// TwinCAT 3 PLC project TcIotOcppChargingStationPlc
// Title: TwinCAT IoT OCPP Charging Station Sample
// Company: Beckhoff Automation GmbH & Co. KG
// ProjectVersion: 1.0.0.0
// ProgramVersion: 3.1.4026.10
// libraries:
//   Tc2_Standard, * (Beckhoff Automation GmbH)
//   Tc2_System, * (Beckhoff Automation GmbH)
//   Tc2_Utilities, * (Beckhoff Automation GmbH)
//   Tc3_Module, * (Beckhoff Automation GmbH)
//   Tc3_OCPP, * (Beckhoff Automation GmbH)
// project tree:
//   GVLs/ VAR_OCPP.TcGVL, VAR_Param.TcGVL
//   / PlcTask.TcTTO
//   POUs/ FB_ConnectorSim.TcPOU, MAIN.TcPOU
//   POUs/OCPP/ FB_Connector.TcPOU, FB_ConnectorMeter.TcPOU, FB_MeterValue.TcPOU, FB_SampleValue.TcPOU, FB_Station.TcPOU, FB_StationMeter.TcPOU
// real-time tasks:
//   TASK PlcTask: cycle T#10ms, priority 20, ADS port 350

CONFIGURATION TcIotOcppChargingStationPlc
    RESOURCE PLC ON TwinCAT3
        TASK PlcTask(INTERVAL := T#10ms, PRIORITY := 20);
        PROGRAM MAIN WITH PlcTask : MAIN;
    END_RESOURCE
END_CONFIGURATION

// ---- GVLs/VAR_OCPP.TcGVL
{attribute 'qualified_only'}
VAR_GLOBAL
	stClientParam : ST_OCPP1_ClientParam := (
		//nOID : OTCID := 0; // ObjectID of the TcIotOcpp Client Object (0 to create a new instance).
		nTaskOID := 0, // ObjectId of the Task whose shall execute the client (0 to use I/O Idle Task)
		sHost := 'localhost', // Defines the server-address by host-name, domain-name or IP-address.
		nPort := 8080, // Defines the server-port.
		sPath := 'ocpp', // Defines the server-path.
		sIdentity := 'Test01', // Defines the client-identity (and user-id).
		eAuthMode := E_OCPP1_AuthenticationMode.Basic, // Defines an optional authentication-mode.
		sAuthKey := 'abcdef', // Defines an optional authentication key.
		eEncryptionMode := E_OCPP_EncryptionMode.None, // Defines an optional encryption mode.
		eTraceLevel := TcTraceLevel.tlVerbose); // Defines the maximum trace level of ADS log messages.

	stOptions : ST_OCPP1_ClientOptions := (
		bAllowOfflineTxForUnknownId := FALSE, // Whether Unknown Offline Authorization is enabled.
		bAuthListEnabled := FALSE, // Whether the Local Authorization List is enabled.
		bAuthCacheEnabled := FALSE, // Whether the Authorization Cache is enabled.
		bLocalAuthOffline := FALSE, // Whether the Charge Point, when offline, will start a transaction for locally-authorized identifiers.
		bLocalPreAuth := FALSE); // Whether the Charge Point, when online, will start a transaction for locally-authorized identifiers without waiting for an response from the Central System.

	stSettings : ST_OCPP1_ClientSettings := (
		nTransactionMessageAttempts := 5, // How often the Charge Point should try to submit a transaction-related message when the Central System fails to process it.
		nTransactionMessageRetryInterval := 5); // [s] How long the Charge Point should wait before resubmitting a transaction-related message that the Central System failed to process.

	stBootInfo : ST_OCPP1_ClientBootInfo := (
		sChargePointModel := 'TcIotOcppStation', // Required. This contains a value that identifies the model of the ChargePoint.
		sChargePointVendor := 'Beckhoff Automation', // Required. This contains a value that identifies the vendor of the ChargePoint.
		sChargeBoxSerialNumber := '', // Optional. This contains a value that identifies the serial number of the Charge Box inside the Charge Point.
		sChargePointSerialNumber := '', // Optional. This contains a value that identifies the serial number of the Charge Point.
		sFirmwareVersion := '', // Optional. This contains the firmware version of the Charge Point.
		sMeterSerialNumber := '', // Optional. This contains the serial number of the main electrical meter of the Charge Point.
		sMeterType := ''); // Optional. This contains the type of the main electrical meter of the Charge Point.

	fCurrentOffered1 : REAL := 16.0; // [A] current offered on every phace of connector (11kW)
	fCurrentOffered2 : REAL := 12.0; // [A] current offered on every phace of connector (8kW)
END_VAR

// ---- GVLs/VAR_Param.TcGVL
{attribute 'qualified_only'}
VAR_GLOBAL CONSTANT
	tSamplePeriodic : TIME := T#30S; // Interval of sample periodic meter values in FB_ConnectorMeter
	tSampleClock : TIME := T#60S; // Interval of sample clock meter values in FB_StationMeter
END_VAR

// ---- POUs/MAIN.TcPOU
PROGRAM MAIN
VAR
	// Station/Connectors
	fbStation : FB_Station(stParam := VAR_OCPP.stClientParam);
	fbConnector1 : FB_Connector(nConnectorId := 1, fbStation := fbStation);
	fbConnector2 : FB_Connector(nConnectorId := 2, fbStation := fbStation);
	// MeterValues/SampledValues
	fbStationMeter : FB_StationMeter(fbStation := fbStation);
	fbConnector1Meter : FB_ConnectorMeter(nConnectorId := 1, fbStation := fbStation);
	fbConnector2Meter : FB_ConnectorMeter(nConnectorId := 2, fbStation := fbStation);
	// Simulation
	fbConnector1Sim : FB_ConnectorSim;
	fbConnector2Sim : FB_ConnectorSim;
END_VAR

fbStation.Execute();

fbStationMeter.Execute(fbStation := fbStation);
fbConnector1Meter.Execute(fbConnector := fbConnector1, fCurrentOffered := VAR_OCPP.fCurrentOffered1);
fbConnector2Meter.Execute(fbConnector := fbConnector2, fCurrentOffered := VAR_OCPP.fCurrentOffered2);

fbConnector1Sim(fbConnector := fbConnector1, fCurrentOffered := VAR_OCPP.fCurrentOffered1);
fbConnector2Sim(fbConnector := fbConnector2, fCurrentOffered := VAR_OCPP.fCurrentOffered2);

END_PROGRAM

// ---- POUs/OCPP/FB_Station.TcPOU
FUNCTION_BLOCK FB_Station
VAR_OUTPUT
	bBusy : BOOL;
	bError : BOOL;
	eState : E_OCPP1_ChargePointStatus := E_OCPP1_ChargePointStatus.Available;
	eErrorState : E_OCPP1_ChargePointStatus := E_OCPP1_ChargePointStatus.None;
END_VAR
VAR
	// client
	_oClient : FB_OCPP1_Client(0);
	// connectors
	_arrConnectors : ARRAY[1..Param_OCPP.nConnectorCount] OF POINTER TO FB_Connector;
	_nConnectorCnt : UDINT;
	_nConnectorMax : UDINT;
	// configuration
	_fbConfiguration : FB_OCPP1_Configuration;
	// charging profile
	_fbChargingProfile : FB_OCPP1_ChargingProfile;
	_arrCharging : ARRAY[1..Param_OCPP.nConnectorCount] OF BOOL;
	// reset
	_fbTcRestart : TC_Restart;
	_fbOsRestart : NT_Reboot;
	
	bTest: BOOL;
END_VAR
VAR PERSISTENT
	_bAvailable : BOOL := TRUE;
END_VAR

METHOD INTERNAL AddConnector : BOOL
VAR_INPUT
	nConnectorId : UDINT;
	pConnector : POINTER TO FB_Connector;
END_VAR
IF nConnectorId < 1 OR nConnectorId > Param_OCPP.nConnectorCount THEN
	RETURN; // invalid connector id!
END_IF

IF pConnector = 0 THEN
	RETURN; // invalid pointer to connector!
END_IF

IF _arrConnectors[nConnectorId] <> 0 THEN
	RETURN; // connector id already used!
END_IF

_arrConnectors[nConnectorId] := pConnector;

_nConnectorCnt := _nConnectorCnt + 1;
IF nConnectorId > _nConnectorMax THEN _nConnectorMax := nConnectorId; END_IF

AddConnector := TRUE;
END_METHOD

PROPERTY Available : BOOL
GET
Available := _oClient.IsConnected
	AND eState <> E_OCPP1_ChargePointStatus.Unavailable
	AND eState <> E_OCPP1_ChargePointStatus.Faulted;
END_GET
END_PROPERTY

PROPERTY INTERNAL Client : POINTER TO FB_OCPP1_Client
GET
Client := ADR(_oClient);
END_GET
END_PROPERTY

METHOD PRIVATE Configuration : BOOL
VAR_STAT
	sValue : T_OCPP1_ConfigValue;
	nValue : UDINT;
END_VAR
IF _fbConfiguration.HasChanged(E_OCPP1_ConfigKey.HeartbeatInterval) THEN
	sValue := _fbConfiguration.GetValue(E_OCPP1_ConfigKey.HeartbeatInterval);
	_oClient.HeartbeatInterval := UDINT_TO_TIME(STRING_TO_UDINT(sValue)*1000);
END_IF
END_METHOD

METHOD Execute : BOOL
VAR
	nIdx : UDINT;
	eAction : E_OCPP1_Action;
	mPeriod : ST_OCPP1_ChargingSchedulePeriod;
END_VAR
_oClient.Execute(TRUE);
bBusy := _oClient.bBusy;

IF _oClient.bError THEN
	bError := TRUE;
	eErrorState := eState;
	eState := E_OCPP1_ChargePointStatus.Faulted;
END_IF

// ================================================================================
// Execute Connectors and apply Charging Profile

FOR nIdx := 1 TO Param_OCPP.nConnectorCount DO
	_arrConnectors[nIdx]^.Execute();
	_arrCharging[nIdx] := _arrConnectors[nIdx]^.bCharging;
END_FOR

_fbChargingProfile.Execute(_arrCharging, _oClient);

FOR nIdx := 1 TO Param_OCPP.nConnectorCount DO
	_fbChargingProfile.GetCurrentPeriod(nIdx, mPeriod);
	_arrConnectors[nIdx]^.SetChargingSchedulePeriod(mPeriod);
END_FOR

// ================================================================================
// State machine of Charging Station

CASE eState OF
	E_OCPP1_ChargePointStatus.Available: // Operative
		IF NOT _bAvailable THEN
			eState := E_OCPP1_ChargePointStatus.Unavailable;
		END_IF

	E_OCPP1_ChargePointStatus.Unavailable: // Inoperative, e.g. as result of a ChangeAvailability command.
		IF _bAvailable THEN
			eState := E_OCPP1_ChargePointStatus.Available;
		END_IF

	E_OCPP1_ChargePointStatus.Faulted: // Inoperative, when charger or connector has reported an error and is not available for energy delivery.

ELSE
	bError := TRUE;
	eErrorState := eState;
	eState := E_OCPP1_ChargePointStatus.Faulted;
END_CASE

// ================================================================================
// Send status of Charging Station

SendStatusNotification();

// ================================================================================
// Receive requests from Management System

IF _oClient.PollRequest(eAction => eAction) THEN
	CASE eAction OF
		// Core
		E_OCPP1_Action.RemoteStartTransaction:
			RecvRemoteStartTransaction();
		E_OCPP1_Action.RemoteStopTransaction:
			RecvRemoteStopTransaction();
		E_OCPP1_Action.ChangeAvailability:
			RecvChangeAvailability();
		E_OCPP1_Action.UnlockConnector:
			RecvUnlockConnector();
		E_OCPP1_Action.ChangeConfiguration:
			_fbConfiguration.Execute(_oClient);
		E_OCPP1_Action.GetConfiguration:
			_fbConfiguration.Execute(_oClient);
		//E_OCPP1_Action.ClearCache
		E_OCPP1_Action.Reset:
			RecvReset();
		// Remote Trigger
		E_OCPP1_Action.TriggerMessage:
			RecvTriggerMessage();
		// Reservation
		E_OCPP1_Action.ReserveNow:
			RecvReserveNow();
		E_OCPP1_Action.CancelReservation:
			RecvReserveCancel();
		// Smart Charging
		E_OCPP1_Action.SetChargingProfile:
			_fbChargingProfile.Execute(_arrCharging, _oClient);
		E_OCPP1_Action.GetCompositeSchedule:
			_fbChargingProfile.Execute(_arrCharging, _oClient);
		E_OCPP1_Action.ClearChargingProfile:
			_fbChargingProfile.Execute(_arrCharging, _oClient);
		// Authentication
		//E_OCPP1_Action.GetLocalListVersion
		//E_OCPP1_Action.SendLocalList
		// Firmware
		//E_OCPP1_Action.GetDiagnostics
		//E_OCPP1_Action.UpdateFirmware
		// Vendor
		E_OCPP1_Action.DataTransfer:
			RecvDataTransfer();
		// Security
		//E_OCPP1_Action.ExtendedTriggerMessage
		//E_OCPP1_Action.GetLog
		//E_OCPP1_Action.GetInstalledCertificateIds
		//E_OCPP1_Action.CertificateSigned
		//E_OCPP1_Action.SignCertificate
		//E_OCPP1_Action.InstallCertificate
		//E_OCPP1_Action.DeleteCertificate
		//E_OCPP1_Action.SignedUpdateFirmware
	ELSE
		// TODO response
	END_CASE
END_IF

// ================================================================================
// Additional functionalities

_fbTcRestart(RESTART := FALSE);
_fbOsRestart(START := FALSE);

Configuration();
SendDataTransfer();
END_METHOD

METHOD FB_Init : BOOL
VAR_INPUT
	bInitRetains : BOOL; // if TRUE, the retain variables are initialized (warm start / cold start)
	bInCopyCode : BOOL;  // if TRUE, the instance afterwards gets moved into the copy code (online change)

	stParam :  REFERENCE TO ST_OCPP1_ClientParam; // Parameter to define the OCPP WebSocket connection.
END_VAR
IF bInCopyCode THEN RETURN; END_IF

IF NOT __ISVALIDREF(stParam) THEN RETURN; END_IF

FB_Init := Init(stParam);
END_METHOD

METHOD Init : BOOL
VAR_INPUT
	stParam : REFERENCE TO ST_OCPP1_ClientParam; // Parameter to define the OCPP WebSocket connection.
END_VAR
Init := _oClient.Init(stParam);

_oClient.InitOptions(VAR_OCPP.stOptions);
_oClient.InitSettings(VAR_OCPP.stSettings);
_oClient.InitBootInfo(VAR_OCPP.stBootInfo);

_fbConfiguration.InitStandard();
_fbConfiguration.InitKeyValue(E_OCPP1_ConfigKey.HeartbeatInterval, UDINT_TO_STRING(TIME_TO_UDINT(_oClient.HeartbeatInterval)/1000), FALSE);
END_METHOD

PROPERTY IsConnected : BOOL
GET
IsConnected := _oClient.IsConnected;
END_GET
END_PROPERTY

METHOD PRIVATE RecvChangeAvailability : BOOL
VAR_STAT
	hRecvId : T_OCPP_MessageId;
	nConnectorId : UDINT; // The id of the connector for which availability needs to change.
	eType : E_OCPP1_AvailabilityType; // This contains the type of availability change that the Charge Point should perform.
	eStatus : E_OCPP1_AvailabilityStatus; // This indicates whether the Charge Point is able to perform the availability change.
END_VAR
// Central System can request a Charge Point to change its availability
// - A Charge Point is considered available ("operative") when it is charging or ready for charging
// - A Charge Point is considered unavailable when it does not allow any charging
IF _oClient.RecvChangeAvailability(hMessageId=> hRecvId, nConnectorId=> nConnectorId, eType=> eType) THEN
	eStatus := E_OCPP1_AvailabilityStatus.Rejected;
	IF nConnectorId = 0 THEN
		CASE eType OF
			E_OCPP1_AvailabilityType.Operative:
				_bAvailable := TRUE;
				eStatus := E_OCPP1_AvailabilityStatus.Accepted;
			E_OCPP1_AvailabilityType.Inoperative:
				_bAvailable := FALSE;
				eStatus := E_OCPP1_AvailabilityStatus.Accepted;
		END_CASE
		FOR nConnectorId := 1 TO _nConnectorMax DO
			IF _arrConnectors[nConnectorId] <> 0 THEN
				_arrConnectors[nConnectorId]^.ChangeAvailability(eType:= eType, eStatus=> eStatus);
			END_IF
		END_FOR
	ELSE
		IF _arrConnectors[nConnectorId] <> 0 THEN
			IF _arrConnectors[nConnectorId]^.ChangeAvailability(eType:= eType, eStatus=> eStatus) THEN
		 		eStatus := E_OCPP1_AvailabilityStatus.Accepted;
			END_IF
		END_IF
	END_IF
	_oClient.RespChangeAvailability(hMessageId:= hRecvId, eStatus:= eStatus);
END_IF
END_METHOD

METHOD RecvDataTransfer : BOOL
VAR_STAT
	hRecvId : T_OCPP_MessageId;
	sVendorId : STRING(255); 
	sMessageId : STRING(63); 
	sData : T_OCPP1_DataTransferData; 
END_VAR
IF _oClient.RecvDataTransfer(hMessageId => hRecvId, sVendorId=> sVendorId, sMessageId=> sMessageId, sData := sData) THEN
	IF sVendorId <> 'Beckhoff Automation' THEN
		_oClient.RespDataTransfer(hRecvId, eStatus := E_OCPP1_DataTransferStatus.UnknownVendorId);
	ELSIF sMessageId <> 'DataTransfer' THEN
		_oClient.RespDataTransfer(hRecvId, eStatus := E_OCPP1_DataTransferStatus.UnknownMessageId);
	ELSE
		_oClient.RespDataTransfer(hRecvId, eStatus := E_OCPP1_DataTransferStatus.Accepted);
	END_IF
END_IF
END_METHOD

METHOD PRIVATE RecvRemoteStartTransaction : BOOL
VAR
	hRecvId : T_OCPP_MessageId;
	nConnectorId : UDINT; // Number of the connector on which to start the transaction.
	sIdTag : T_OCPP1_IdToken; // The identifier that Charge Point must use to start a transaction.
	eStatus : E_OCPP1_RemoteStartStopStatus; // Status indicating whether Charge Point accepts the request to start a transaction.
END_VAR
// Central System can request a Charge Point to start a transaction
// - Enable a operator to help a driver that has problems starting a transaction
// - Enable mobile apps to control charging transactions via the Central System
IF _oClient.RecvRemoteStartTransaction(hMessageId=> hRecvId, nConnectorId=> nConnectorId, sIdToken=> sIdTag) THEN
	eStatus := E_OCPP1_RemoteStartStopStatus.Rejected;
	IF nConnectorId = 0 AND _nConnectorCnt = 1 THEN
		nConnectorId := 1; // Workaround optional ConnectorId
	END_IF
	IF nConnectorId <> 0 THEN
		IF _arrConnectors[nConnectorId] <> 0 THEN
			IF _arrConnectors[nConnectorId]^.RemoteStartTransaction(sIdTag) THEN
		 		eStatus := E_OCPP1_RemoteStartStopStatus.Accepted;
			END_IF
		END_IF
	END_IF
	_oClient.RespRemoteStartTransaction(hMessageId:= hRecvId, eStatus:= eStatus);
END_IF
END_METHOD

METHOD PRIVATE RecvRemoteStopTransaction : BOOL
VAR
	hRecvId : T_OCPP_MessageId;
	nConnectorId : UDINT; // This identifies which connector of the Charge Point is used.
	eStatus : E_OCPP1_RemoteStartStopStatus; // Status indicating whether Charge Point accepts the request to stop a transaction.
END_VAR
// Central System can request a Charge Point to stop a transaction
// - Enable a operator to help a driver that has problems stopping a transaction
// - Enable mobile apps to control charging transactions via the Central System
IF _oClient.RecvRemoteStopTransaction(hMessageId=> hRecvId, nConnectorId=> nConnectorId) THEN
	eStatus := E_OCPP1_RemoteStartStopStatus.Rejected;
	IF nConnectorId > 0 AND nConnectorId <= _nConnectorMax THEN
		IF _arrConnectors[nConnectorId] <> 0 THEN
			IF _arrConnectors[nConnectorId]^.RemoteStopTransaction() THEN
				eStatus := E_OCPP1_RemoteStartStopStatus.Accepted;

			END_IF
		END_IF
	END_IF
	_oClient.RespRemoteStopTransaction(hMessageId:= hRecvId, eStatus:= eStatus);
END_IF
END_METHOD

METHOD RecvReserveCancel : BOOL
VAR
	hRecvId : T_OCPP_MessageId;
	nReservationId : UDINT;
	nConnectorId : UDINT;
	eStatus : E_OCPP1_CancelReservationStatus;
END_VAR
IF _oClient.RecvCancelReservation(hMessageId => hRecvId, nReservationId => nReservationId) THEN
	eStatus := E_OCPP1_CancelReservationStatus.Rejected;
	FOR nConnectorId := 1 TO Param_OCPP.nConnectorCount DO
		IF _arrConnectors[nConnectorId] <> 0 THEN
			IF _arrConnectors[nConnectorId]^.ReserveCancel(nReservationId) THEN
				eStatus := E_OCPP1_CancelReservationStatus.Accepted;
				EXIT;
			END_IF
		END_IF
	END_FOR
	_oClient.RespCancelReservation(hRecvId, eStatus);	
END_IF
END_METHOD

METHOD PRIVATE RecvReserveNow : BOOL
VAR
	hRecvId : T_OCPP_MessageId;
	nConnectorId : UDINT;
	sIdTag: T_OCPP1_IdToken;
	nReservationId: UDINT;
	eStatus: E_OCPP1_ReservationStatus;
END_VAR
IF _oClient.RecvReserveNow(hMessageId => hRecvId, nConnectorId => nConnectorId, sIdTag => sIdTag, nReservationId => nReservationId) THEN
	eStatus := E_OCPP1_ReservationStatus.Rejected;
	IF nConnectorId <> 0 THEN
		IF _arrConnectors[nConnectorId] <> 0 THEN
			IF _arrConnectors[nConnectorId]^.Reserve(sIdTag, nReservationId) THEN
				eStatus := E_OCPP1_ReservationStatus.Accepted;
			ELSE
				eStatus := E_OCPP1_ReservationStatus.Occupied;
			END_IF
		END_IF
	END_IF
	// TODO #183271
	// _oClient.SendResponse(hMessageId:= hRecvId, E_OCPP1_Action.ReserveNow, SIZEOF(mRes), ADR(mRes));
END_IF
END_METHOD

METHOD RecvReset : BOOL
VAR
	hRecvId : T_OCPP_MessageId;
	eType : E_OCPP1_ResetType;
END_VAR
// Central System can request a Charge Point to reset itself
// - At receipt of a soft reset, the Charge Point shall stop ongoing transactions
// - At receipt of a hard reset the Charge Point shall restart (all) the hardware, not required to stop ongoing transaction
IF _oClient.RecvReset(hMessageId=> hRecvId, eType=> eType) THEN
		IF eType = E_OCPP1_ResetType.Soft THEN
			_oClient.RespReset(hMessageId:= hRecvId, eStatus:= E_OCPP1_ResetStatus.Accepted);
			_fbTcRestart(RESTART := TRUE);
		ELSIF eType = E_OCPP1_ResetType.Hard THEN
			_oClient.RespReset(hMessageId:= hRecvId, eStatus:= E_OCPP1_ResetStatus.Accepted);
			_fbOsRestarT(START := TRUE);
		ELSE
			_oClient.RespReset(hMessageId:= hRecvId, eStatus:= E_OCPP1_ResetStatus.Rejected);
		END_IF
END_IF
END_METHOD

METHOD RecvTriggerMessage : BOOL
VAR_STAT
	hRecvId : T_OCPP_MessageId;
	eRequestedMessage: E_OCPP1_MessageTrigger;
	nConnectorId : UDINT;
	eStatus: E_OCPP1_TriggerMessageStatus;
END_VAR
hRecvId := '';
IF _oClient.RecvTriggerMessage(hMessageId => hRecvId, eRequestedMessage => eRequestedMessage) THEN
	nConnectorId := 1; // TODO #183270
	eStatus := E_OCPP1_TriggerMessageStatus.Rejected;
	IF nConnectorId <> 0 THEN
		IF _arrConnectors[nConnectorId] <> 0 THEN
			IF _arrConnectors[nConnectorId]^.TriggerMessage(eRequestedMessage) THEN
		 		eStatus := E_OCPP1_TriggerMessageStatus.Accepted;
			END_IF
		END_IF
	END_IF
	_oClient.RespTriggerMessage(hRecvId, eStatus);
END_IF
END_METHOD

METHOD PRIVATE RecvUnlockConnector : BOOL
VAR
	hRecvId : T_OCPP_MessageId;
	nConnectorId : UDINT; // This contains the identifier of the connector to be unlocked.
	eStatus : E_OCPP1_UnlockStatus; // This indicates whether the Charge Point has unlocked the connector.
END_VAR
// Central System can request a Charge Point to unlock a connector
// - Help drivers that have problems unplugging their cable from the Charge Point in case of malfunction
IF _oClient.RecvUnlockConnector(hMessageId=> hRecvId, nConnectorId=> nConnectorId) THEN
	eStatus := E_OCPP1_UnlockStatus.UnlockFailed;
	IF nConnectorId <> 0 THEN
		IF _arrConnectors[nConnectorId] <> 0 THEN
			IF _arrConnectors[nConnectorId]^.UnlockConnector() THEN
		 		eStatus := E_OCPP1_UnlockStatus.Unlocked;
			END_IF
		END_IF
	END_IF
	_oClient.RespUnlockConnector(hMessageId:= hRecvId, eStatus:= eStatus);
END_IF
END_METHOD

METHOD SendDataTransfer : BOOL
VAR_STAT
	bSend : BOOL;
END_VAR
IF bSend THEN
	IF _oClient.SendDataTransfer('Beckhoff Automation', 'Hello World', '{"Hello":"World"}') THEN
		bSend := FALSE;
	END_IF
END_IF
END_METHOD

METHOD PRIVATE SendStatusNotification : BOOL
VAR_INST
	bSend : BOOL;
	eSend : E_OCPP1_ChargePointStatus;
	eLast : E_OCPP1_ChargePointStatus;
END_VAR
// Keep the charging station informed about the charger status
// - Sends a notification to Server and inform about a status change or an error
// - Memorize latest state and send if connected, otherwise keep it until reconnected
IF NOT bSend AND eState <> eLast THEN
	bSend := (eState <> E_OCPP1_ChargePointStatus.None);
	eSend := eState;
END_IF
IF bSend AND _oClient.IsConnected THEN
	IF _oClient.SendStatusNotification(0, E_OCPP1_ChargePointError.NoError, eState) THEN
		bSend := FALSE;
		eLast := eState;
	END_IF
END_IF
END_METHOD

END_FUNCTION_BLOCK

// ---- POUs/OCPP/FB_Connector.TcPOU
FUNCTION_BLOCK FB_Connector
VAR_INPUT
	bOperative : BOOL; // Operative and ready for energy delivery
	sIdTag : T_OCPP1_IdToken; // Token of id tag

	bAuth : BOOL; // Request to authorize identity
	bStart : BOOL; // Request to start a transaction
	bStop : BOOL; // Request to stop a transaction

	bConnected : BOOL; // Plug is inserted
	bLocked : BOOL; // Cable is locked
	bOffering : BOOL; // Supply is offering energy
	bCharging : BOOL; // Vehicle is taking energy
	nEnergyMeter : UDINT; // Accumulated meter value in Wh of the connector
END_VAR
VAR_OUTPUT
	fChargeLimit : REAL; // [A] Charging rate limit of current offered on every phace of connector
	bLock : BOOL; // Request to lock cable (on supply and/or vehicle)
	bSupply : BOOL; // Request to supply energy to vehicle
	bBusy : BOOL;
	bError : BOOL;
	eState : E_OCPP1_ChargePointStatus := E_OCPP1_ChargePointStatus.Available;
	eErrorAction : E_OCPP1_Action := E_OCPP1_Action.None;
	eErrorState : E_OCPP1_ChargePointStatus := E_OCPP1_ChargePointStatus.None;
	eAuthStatus : E_OCPP1_AuthorizationStatus := E_OCPP1_AuthorizationStatus.None;
	eStopReason : E_OCPP1_Reason := E_OCPP1_Reason.None; // Reason why the transaction was stopped.
END_VAR
VAR
	// id
	_nConnectorId : UDINT;
	// client
	_pClient : POINTER TO FB_OCPP1_Client;
	// memory
	_sIdTag : T_OCPP1_IdToken;
	// trigger
	_trigAuth : R_TRIG;
	_bAuth : BOOL;
	_trigLocalStart : R_TRIG;
	_bStart : BOOL;
	_trigLocalStop : R_TRIG;
	_bStop : BOOL;
	// transaction
	_bTransActive : BOOL;
	// reservation
	_bReserved : BOOL;
	_sReserveId : T_OCPP1_IdToken;
	_nReserveId : UDINT;
END_VAR
VAR PERSISTENT
	_bAvailable : BOOL := TRUE;
END_VAR

PROPERTY Available : BOOL
GET
Available := _pClient <> 0 AND _pClient^.IsConnected
	AND eState <> E_OCPP1_ChargePointStatus.Unavailable
	AND eState <> E_OCPP1_ChargePointStatus.Faulted;
END_GET
END_PROPERTY

METHOD INTERNAL ChangeAvailability : BOOL
VAR_INPUT
	eType : E_OCPP1_AvailabilityType; // This contains the type of availability change that the Charge Point should perform.
END_VAR
VAR_OUTPUT
	eStatus : E_OCPP1_AvailabilityStatus; // This indicates whether the Charge Point is able to perform the availability change.
END_VAR
CASE eType OF
	E_OCPP1_AvailabilityType.Operative:
		_bAvailable := TRUE;
		eStatus := E_OCPP1_AvailabilityStatus.Accepted;
		ChangeAvailability := TRUE;
	E_OCPP1_AvailabilityType.Inoperative:
		_bAvailable := FALSE;
		CASE eState OF
			E_OCPP1_ChargePointStatus.Available:
				eStatus := E_OCPP1_AvailabilityStatus.Accepted;
			E_OCPP1_ChargePointStatus.Preparing:
				eStatus := E_OCPP1_AvailabilityStatus.Scheduled;
			E_OCPP1_ChargePointStatus.Charging:
				eStatus := E_OCPP1_AvailabilityStatus.Scheduled;
			E_OCPP1_ChargePointStatus.SuspendedEVSE:
				eStatus := E_OCPP1_AvailabilityStatus.Scheduled;
			E_OCPP1_ChargePointStatus.SuspendedEV:
				eStatus := E_OCPP1_AvailabilityStatus.Scheduled;
			E_OCPP1_ChargePointStatus.Finishing:
				eStatus := E_OCPP1_AvailabilityStatus.Accepted;
			E_OCPP1_ChargePointStatus.Reserved:
				eStatus := E_OCPP1_AvailabilityStatus.Accepted;
			E_OCPP1_ChargePointStatus.Unavailable:
				eStatus := E_OCPP1_AvailabilityStatus.Accepted;
			E_OCPP1_ChargePointStatus.Faulted:
				eStatus := E_OCPP1_AvailabilityStatus.Accepted;
		END_CASE
		ChangeAvailability := TRUE;
ELSE
	eStatus := E_OCPP1_AvailabilityStatus.Rejected;
	ChangeAvailability := FALSE;
END_CASE
END_METHOD

METHOD Execute : BOOL
IF _pClient <> 0 THEN
	bBusy := _pClient^.bBusy;
	IF _pClient^.bError AND NOT bError THEN
		bError := _pClient^.bError;
		eErrorAction := _pClient^.eErrorAction;
		eErrorState := eState;
		eState := E_OCPP1_ChargePointStatus.Faulted;
	END_IF
ELSE
	bError := TRUE;
	eErrorState := E_OCPP1_ChargePointStatus.None;
	RETURN;
END_IF

// ================================================================================
// Trigger

_trigAuth(CLK := bAuth);
IF _trigAuth.Q THEN
	eAuthStatus := E_OCPP1_AuthorizationStatus.None;
	_bAuth := TRUE;
	_sIdTag := sIdTag;
END_IF

_trigLocalStart(CLK := bStart AND bConnected);
IF _trigLocalStart.Q AND NOT _bStart
	AND_THEN (eState = E_OCPP1_ChargePointStatus.Available
		OR eState = E_OCPP1_ChargePointStatus.Preparing
		OR eState = E_OCPP1_ChargePointStatus.Finishing)
THEN
	IF eAuthStatus <> E_OCPP1_AuthorizationStatus.Accepted THEN
		eAuthStatus := E_OCPP1_AuthorizationStatus.None;
		_bAuth := TRUE;
		_sIdTag := sIdTag;
	END_IF
	_bStart := TRUE;
END_IF

_trigLocalStop(CLK := bStop AND bSupply);
IF _trigLocalStop.Q AND NOT _bStop
	AND_THEN (eState = E_OCPP1_ChargePointStatus.Charging
		OR eState = E_OCPP1_ChargePointStatus.SuspendedEVSE
		OR eState = E_OCPP1_ChargePointStatus.SuspendedEV)
THEN
	IF eAuthStatus <> E_OCPP1_AuthorizationStatus.Accepted THEN
		eAuthStatus := E_OCPP1_AuthorizationStatus.None;
		_bAuth := TRUE;
		_sIdTag := sIdTag;
	END_IF
	eStopReason := E_OCPP1_Reason.Local;
	_bStop := TRUE;
END_IF

// ================================================================================
// State machine of connector

CASE eState OF
	E_OCPP1_ChargePointStatus.Available: // When a connector becomes available for a new user. (Operative)

		// Transition A2 ==> Preparing
		// Transition A3, A4, A5 ==> Preparing and then following transitions
		// - Usage is initiated (e.g. insert plug, bay occupancy detection, present idTag, push start button, receipt of a RemoteStartTransaction request)
		IF bConnected THEN
			eState := E_OCPP1_ChargePointStatus.Preparing;
		END_IF

		// Transition A7 ==> Reserved
		// - A ReserveNow message is received that reserves the connector
		IF _bReserved THEN
			eState := E_OCPP1_ChargePointStatus.Reserved;
		END_IF

		// Transition A8 ==> Unavailable
		// - A ChangeAvailability message is received that sets the connector to Unavailable
		IF NOT _bAvailable THEN
			eState := E_OCPP1_ChargePointStatus.Unavailable;
		END_IF

	E_OCPP1_ChargePointStatus.Preparing: // When a connector becomes no longer available for a new user but there is no ongoing transaction. (Operative)

		// Transition B1 ==> Available
		// - Intended usage is ended (e.g. plug removed, bay no longer occupied, second presentation of idTag, time out on expected user action)
		IF NOT bConnected THEN
			eState := E_OCPP1_ChargePointStatus.Available;
		END_IF

		// Connected cable => lock cable
		IF _bStart AND bConnected THEN
			// Authorize the operation
			// - Before the owner of a vehicle can start/stop charging, the Charge Point has to authorize the operation
			IF eAuthStatus = E_OCPP1_AuthorizationStatus.Accepted THEN
				bLock := TRUE;
			ELSIF eAuthStatus <> E_OCPP1_AuthorizationStatus.None THEN
				bLock := FALSE;
				eState := E_OCPP1_ChargePointStatus.Finishing;
			END_IF
		ELSE
			bLock := FALSE;
		END_IF

		// Locked cable => supply energy
		IF bLock AND bLocked THEN
			// Authorize the operation
			// - Before the owner of a vehicle can start/stop charging, the Charge Point has to authorize the operation
			IF eAuthStatus = E_OCPP1_AuthorizationStatus.Accepted THEN
				bSupply := TRUE;
			ELSIF eAuthStatus <> E_OCPP1_AuthorizationStatus.None THEN
				bSupply := FALSE;
				eState := E_OCPP1_ChargePointStatus.Finishing;
			END_IF
		ELSE
			bSupply := FALSE;
		END_IF

		IF bSupply THEN
			// Transition B5 ==> SuspendedEVSE
			// - All prerequisites for charging are met but EVSE does not allow charging
			IF NOT bOffering THEN
				eState := E_OCPP1_ChargePointStatus.SuspendedEVSE;
				_bStart := FALSE;
			// Transition B4 ==> SuspendedEV
			// - All prerequisites for charging are met but EV does not start charging
			ELSIF NOT bCharging THEN
				eState := E_OCPP1_ChargePointStatus.SuspendedEV;
				_bStart := FALSE;
			// Transition B3 ==> Charging
			// - All prerequisites for charging are met and charging process starts
			ELSE // bOffering AND bCharging
				eState := E_OCPP1_ChargePointStatus.Charging;
				_bStart := FALSE;
			END_IF
		END_IF

		// Transition B6 ==> Finishing
		// - Timed out. Usage was initiated (e.g. insert plug, bay occupancy detection), but idTag not presented within timeout.
		// ==> TODO

	E_OCPP1_ChargePointStatus.Charging: // When the contactor of a connector closes, allowing the vehicle to charge. (Operative)

		// Transition C1 ==> Available
		// - Charging session ends while no user action is required (e.g. fixed cable was removed on EV side)
		IF NOT bConnected THEN
			bLock := FALSE;
			bSupply := FALSE;
			eState := E_OCPP1_ChargePointStatus.Available;
			eStopReason := E_OCPP1_Reason.EVDisconnected;
			_bStop := TRUE;
		END_IF

		// Transition C4 ==> SuspendedEV
		// - Charging stops upon EV request (e.g. S2 is opened)
		IF NOT bCharging THEN
			eState := E_OCPP1_ChargePointStatus.SuspendedEV;
		END_IF

		// Transition C5 ==> SuspendedEVSE
		// - Charging stops upon EVSE request (e.g. smart charging restriction, transaction is invalidated by the AuthorizationStatus in a StartTransaction response)
		IF NOT bOffering THEN
			eState := E_OCPP1_ChargePointStatus.SuspendedEVSE;
		END_IF

		// Transition C6 ==> Finishing
		// Transition C8 ==> Finishing and then Unavailable
		// - Transaction is stopped by user or a Remote Stop Transaction message and further user action is required (e.g. remove cable, leave parking bay)
		IF _bStop THEN
			bSupply := FALSE;
			eState := E_OCPP1_ChargePointStatus.Finishing;
		END_IF
		IF eAuthStatus <> E_OCPP1_AuthorizationStatus.Accepted THEN
			bSupply := FALSE;
			eState := E_OCPP1_ChargePointStatus.Finishing;
			eStopReason := E_OCPP1_Reason.DeAuthorized;
			_bStop := TRUE;
		END_IF

	E_OCPP1_ChargePointStatus.SuspendedEVSE: // When the EV is connected to the EVSE but the EVSE is not offering energy to the EV. (Operative)

		// Transition E1 ==> Available
		// - Charging session ends while no user action is required
		IF NOT bConnected THEN
			bLock := FALSE;
			bSupply := FALSE;
			eState := E_OCPP1_ChargePointStatus.Available;
			eStopReason := E_OCPP1_Reason.EVDisconnected;
			_bStop := TRUE;
		END_IF

		// Transition E3 ==> Charging
		// - Charging resumes because the EVSE restriction is lifted
		IF bOffering AND bCharging THEN
			eState := E_OCPP1_ChargePointStatus.Charging;
		END_IF

		// Transition E4 ==> SuspendedEV
		// - The EVSE restriction is lifted but the EV does not start charging
		IF bOffering AND NOT bCharging THEN
			eState := E_OCPP1_ChargePointStatus.SuspendedEV;
		END_IF

		// Transition E6 ==> Finishing
		// Transition E8 ==> Finishing and then Unavailable
		// - Transaction is stopped and further user action is required
		IF _bStop THEN
			bSupply := FALSE;
			eState := E_OCPP1_ChargePointStatus.Finishing;
		END_IF
		IF eAuthStatus <> E_OCPP1_AuthorizationStatus.Accepted THEN
			eState := E_OCPP1_ChargePointStatus.Finishing;
			bSupply := FALSE;
			eStopReason := E_OCPP1_Reason.DeAuthorized;
			_bStop := TRUE;
		END_IF

	E_OCPP1_ChargePointStatus.SuspendedEV: // When the EV is connected to the EVSE and the EVSE is offering energy but the EV is not taking any energy. (Operative)

		// Transition D1 ==> Available
		// - Charging session ends while no user action is required
		IF NOT bConnected THEN
			bLock := FALSE;
			bSupply := FALSE;
			eState := E_OCPP1_ChargePointStatus.Available;
			eStopReason := E_OCPP1_Reason.EVDisconnected;
			_bStop := TRUE;
		END_IF

		// Transition D3 ==> Charging
		// - Charging resumes upon request of the EV (e.g. S2 is closed)
		IF bOffering AND bCharging THEN
			eState := E_OCPP1_ChargePointStatus.Charging;
		END_IF

		// Transition D5 ==> SuspendedEVSE
		// - Charging is suspended by EVSE (e.g. due to a smart charging restriction)
		IF NOT bOffering THEN
			eState := E_OCPP1_ChargePointStatus.SuspendedEVSE;
		END_IF

		// Transition D6 ==> Finishing
		// Transition D8 ==> Finishing and then Unavailable
		// - Transaction is stopped and further user action is required
		IF _bStop THEN
			bSupply := FALSE;
			eState := E_OCPP1_ChargePointStatus.Finishing;
		END_IF
		IF eAuthStatus <> E_OCPP1_AuthorizationStatus.Accepted THEN
			eState := E_OCPP1_ChargePointStatus.Finishing;
			bSupply := FALSE;
			eStopReason := E_OCPP1_Reason.DeAuthorized;
			_bStop := TRUE;
		END_IF

	E_OCPP1_ChargePointStatus.Finishing: // When a Transaction has stopped at a connector, but the connector is not yet available for a new user. (Operative)

		IF _bStop AND NOT bOffering THEN
			bLock := FALSE;
			_bStop := FALSE;
		END_IF

		// Transition F1 ==> Available
		// - All user actions completed
		IF NOT bConnected THEN
			eState := E_OCPP1_ChargePointStatus.Available;
		END_IF

		// Transition F2 ==> Preparing
		// - User restart charging session (e.g. reconnects cable, presents idTag again), thereby creating a new Transaction
		IF _bStart THEN
			// Authorize the operation
			// - Before the owner of a vehicle can start/stop charging, the Charge Point has to authorize the operation
			IF eAuthStatus = E_OCPP1_AuthorizationStatus.Accepted THEN
				eState := E_OCPP1_ChargePointStatus.Preparing;
			ELSE
				_bStart := FALSE;
			END_IF
		END_IF

		// Transition F8 ==> Unavailable
		// - All user actions completed and the connector is scheduled to become Unavailable
		IF NOT _bAvailable THEN
			eState := E_OCPP1_ChargePointStatus.Unavailable;
		END_IF

	E_OCPP1_ChargePointStatus.Reserved: // When a Connector becomes reserved as a result of a Reserve Now command. (Operative)

		// Transition G1 ==> Available
		// - Reservation expires or a CancelReservation message is received
		IF NOT _bReserved THEN
			eState := E_OCPP1_ChargePointStatus.Available;
		END_IF

		// Transition G2 ==> Preparing
		// - Reservation identity is presented
		IF _bAuth AND _sIdTag = _sReserveId THEN
			eState := E_OCPP1_ChargePointStatus.Preparing;
			eAuthStatus := E_OCPP1_AuthorizationStatus.Accepted;
			_bStart := TRUE;
		END_IF

		// Transition G8 ==> Unavailable
		// - Reservation expires or a Cancel Reservation message is received and the connector is scheduled to become Unavailable
		// ==> TODO

	E_OCPP1_ChargePointStatus.Unavailable: // When a Connector becomes unavailable as the result of a ChangeAvailability command or an event upon which the Charge Point transitions to unavailable at its discretion. (Inoperative)

		// Transition H1 ==> Available
		// Transition H2, H3, H4, H4 ==> Available and then following transitions
		// - Connector is set Available by a ChangeAvailability message
		IF _bAvailable THEN
			eState := E_OCPP1_ChargePointStatus.Available;
		END_IF

	E_OCPP1_ChargePointStatus.Faulted: //When a Charge Point or connector has reported an error and is not available for energy delivery . (Inoperative)

		bSupply := FALSE;
		bLock := (bOffering OR bCharging);

		// Transition I1-8
		// - Fault is resolved and status returns to the pre-fault state
		IF NOT (bConnected OR bLocked OR bOffering OR bCharging)  THEN
			eState := E_OCPP1_ChargePointStatus.Available;
			_bAuth := FALSE;
			_bStart := FALSE;
			_bStop := FALSE;
		END_IF

ELSE
	bError := TRUE;
	eErrorState := eState;
	eState := E_OCPP1_ChargePointStatus.Faulted;
END_CASE

// ================================================================================
// Send status of connector
SendAuthorize();
SendStartTransaction();
SendStopTransaction();
SendStatusNotification();
END_METHOD

METHOD FB_Init : BOOL
VAR_INPUT
	bInitRetains : BOOL; // if TRUE, the retain variables are initialized (warm start / cold start)
	bInCopyCode : BOOL;  // if TRUE, the instance afterwards gets moved into the copy code (online change)

	nConnectorId : UDINT;
	fbStation : REFERENCE TO FB_Station;
END_VAR
IF bInCopyCode THEN RETURN; END_IF

IF NOT __ISVALIDREF(fbStation) THEN RETURN; END_IF

FB_Init := Init(nConnectorId, fbStation);
END_METHOD

METHOD Init : BOOL
VAR_INPUT
	nConnectorId : UDINT;
	fbStation : REFERENCE TO FB_Station;
END_VAR
_nConnectorId := nConnectorId;
_pClient := fbStation.Client;

Init := fbStation.AddConnector(_nConnectorId, THIS);
END_METHOD

METHOD INTERNAL RemoteStartTransaction : BOOL
VAR_INPUT
	sIdTag : T_OCPP1_IdToken; // The identifier that Charge Point must use to start a transaction.
END_VAR
_bStart := TRUE;
_sIdTag := sIdTag;

// identifier has already been authorized
eAuthStatus := E_OCPP1_AuthorizationStatus.Accepted;
RemoteStartTransaction := TRUE;
END_METHOD

METHOD INTERNAL RemoteStopTransaction : BOOL
RemoteStopTransaction := StopTransaction(E_OCPP1_Reason.Remote);
END_METHOD

METHOD Reserve : BOOL
VAR_IN_OUT CONSTANT
	sIdTag : T_OCPP1_IdToken;
	nReservationId : UDINT;
END_VAR
IF eState = E_OCPP1_ChargePointStatus.Available THEN
	_bReserved := TRUE;
	_sReserveId := sIdTag;
	_nReserveId := nReservationId;
	Reserve := TRUE;
END_IF
END_METHOD

METHOD ReserveCancel : BOOL
VAR_IN_OUT CONSTANT
	nReservationId : UDINT;
END_VAR
IF _bReserved AND _nReserveId = nReservationId THEN
	_bReserved := FALSE;
	_nReserveId := 0;
	_sReserveId := '';
	ReserveCancel := TRUE;
END_IF
END_METHOD

METHOD PRIVATE SendAuthorize : BOOL
VAR_INST
	eStatus : E_OCPP1_AuthorizationStatus;
END_VAR
// Authorize the operation
// - Before the owner of a vehicle can start/stop charging, the Charge Point has to authorize the operation
IF _bAuth AND _sIdTag <> '' THEN
	IF _pClient^.SendAuthorize(sIdTag := _sIdTag, eStatus=> eStatus) THEN
		_bAuth := FALSE;
		IF NOT _pClient^.bError THEN
			eAuthStatus := eStatus;
		ELSE
			bError := TRUE;
			eErrorState := eState;
			eState := E_OCPP1_ChargePointStatus.Faulted;
			eAuthStatus := E_OCPP1_AuthorizationStatus.Invalid;
		END_IF
	END_IF
END_IF
END_METHOD

METHOD SendHeartbeat : BOOL
VAR_STAT
	hMessageId : UDINT;
(*
	mRequest : ST_OCPP1_HeartbeatReq;
	mResponse: ST_OCPP1_HeartbeatRes;
*)
	nState: INT;
	eError: E_OCPP1_Error;
END_VAR
VAR CONSTANT
	eAction : E_OCPP1_Action := E_OCPP1_Action.Heartbeat;
END_VAR
(*
CASE nState OF
	0:
		IF _pClient^.SendRequest(hMessageId:= hMessageId, eAction:= eAction, nRequest:= SIZEOF(mRequest), pRequest:= ADR(mRequest)) THEN
			nState:=10;
		END_IF
	10:
		IF _pClient^.RecvResponse(hMessageId:=hMessageId , eAction:=eAction , eError:= eError, nResponse:=SIZEOF(mResponse) , pResponse:= ADR(mResponse)) THEN
			nState := 20;
		ELSIF _pClient^.bError THEN
			nState := 20;
		END_IF
	20: 
		SendHeartbeat := TRUE;
		nState := 0; 
END_CASE
*)
END_METHOD

METHOD PRIVATE SendStartTransaction : BOOL
VAR_INST
	trigSend : R_TRIG;
	bSend : BOOL;
	eStatus : E_OCPP1_AuthorizationStatus;
END_VAR
// Start transaction
// - inform about a transaction that has been started
trigSend(CLK := _bStart);
IF trigSend.Q AND NOT _bTransActive THEN
	bSend := TRUE;
	_bTransActive := TRUE;
END_IF
IF bSend THEN
	IF _pClient^.SendStartTransaction(
			sIdTag := _sIdTag,
			nConnectorId := _nConnectorId,
			nMeterStart := nEnergyMeter,
			nReservationId := _nReserveId,
			eStatus=> eStatus)
	THEN
		bSend := FALSE;
		IF NOT _pClient^.bError THEN
			eAuthStatus := eStatus; // TODO Abort a running transaction?
		ELSE
			bError := TRUE;
			eErrorState := eState;
			eState := E_OCPP1_ChargePointStatus.Faulted;
			eAuthStatus := E_OCPP1_AuthorizationStatus.Invalid;
		END_IF
	END_IF
END_IF
END_METHOD

METHOD PRIVATE SendStatusNotification : BOOL
VAR_INST
	bSend : BOOL;
	eSend : E_OCPP1_ChargePointStatus;
	eLast : E_OCPP1_ChargePointStatus;
END_VAR
// Keep the charging station informed about the connector status
// - Sends a notification to Server and inform about a status change or an error
// - Memorize latest state and send if connected, otherwise keep it until reconnected
IF NOT bSend AND eState <> eLast THEN
	bSend := (eState <> E_OCPP1_ChargePointStatus.None);
	eSend := eState;
END_IF
IF bSend AND _pClient^.IsConnected THEN
	IF _pClient^.SendStatusNotification(_nConnectorId, E_OCPP1_ChargePointError.NoError, eSend) THEN
		bSend := FALSE;
		eLast := eState;
	END_IF
END_IF
END_METHOD

METHOD PRIVATE SendStopTransaction : BOOL
VAR_INST
	trigSend : R_TRIG;
	bSend : BOOL;
	eStatus : E_OCPP1_AuthorizationStatus;
END_VAR
// Stop transaction
// - inform about a transaction that has been stopped
trigSend(CLK :=  _bStop);
IF trigSend.Q AND _bTransActive THEN
	bSend := TRUE;
	_bTransActive := FALSE;
END_IF
IF bSend THEN
	IF _pClient^.SendStopTransaction(
			sIdTag := _sIdTag,
			nConnectorId := _nConnectorId,
			nMeterStop := nEnergyMeter,
			eReason := eStopReason,
			eStatus=> eStatus)
	THEN
		bSend := FALSE;
		IF NOT _pClient^.bError THEN
			eAuthStatus := eStatus;
		ELSE
			bError := TRUE;
			eErrorState := eState;
			eState := E_OCPP1_ChargePointStatus.Faulted;
			eAuthStatus := E_OCPP1_AuthorizationStatus.Invalid;
		END_IF
	END_IF
END_IF
END_METHOD

METHOD SetChargingSchedulePeriod : BOOL
VAR_IN_OUT
	mPeriod : ST_OCPP1_ChargingSchedulePeriod;
END_VAR
fChargeLimit := mPeriod.fLimit;
END_METHOD

METHOD INTERNAL StopTransaction : BOOL
VAR_INPUT
	eReason : E_OCPP1_Reason; // This contains the reason why the transaction was stopped.
END_VAR
eStopReason := eReason;
_bStart := FALSE;
_bStop := TRUE;

StopTransaction := TRUE;
END_METHOD

METHOD PUBLIC TriggerMessage : BOOL
VAR_INPUT
	eRequestedMessage : E_OCPP1_MessageTrigger;
END_VAR
CASE eRequestedMessage OF
	//E_OCPP1_MessageTrigger.BootNotification:
	//E_OCPP1_MessageTrigger.DiagnosticsStatusNotification:
	//E_OCPP1_MessageTrigger.FirmwareStatusNotification:
	E_OCPP1_MessageTrigger.Heartbeat:
		TriggerMessage := SendHeartbeat();
	//E_OCPP1_MessageTrigger.MeterValues:

	E_OCPP1_MessageTrigger.StatusNotification:
		TriggerMessage := _pClient^.SendStatusNotification(_nConnectorId, E_OCPP1_ChargePointError.NoError, eState);
END_CASE
END_METHOD

METHOD INTERNAL UnlockConnector : BOOL
CASE eState OF
	E_OCPP1_ChargePointStatus.Preparing:
		StopTransaction(E_OCPP1_Reason.UnlockCommand);
		UnlockConnector := TRUE;
	E_OCPP1_ChargePointStatus.Charging:
		StopTransaction(E_OCPP1_Reason.UnlockCommand);
		UnlockConnector := TRUE;
	E_OCPP1_ChargePointStatus.SuspendedEVSE:
		StopTransaction(E_OCPP1_Reason.UnlockCommand);
		UnlockConnector := TRUE;
	E_OCPP1_ChargePointStatus.SuspendedEV:
		StopTransaction(E_OCPP1_Reason.UnlockCommand);
		UnlockConnector := TRUE;
	E_OCPP1_ChargePointStatus.Finishing:
		StopTransaction(E_OCPP1_Reason.UnlockCommand);
		UnlockConnector := TRUE;
ELSE
	UnlockConnector := FALSE;
END_CASE
END_METHOD

END_FUNCTION_BLOCK

// ---- POUs/OCPP/FB_StationMeter.TcPOU
FUNCTION_BLOCK FB_StationMeter
VAR
	tonSample : TON;
	fbMeter : FB_MeterValue(0, 0);
	fbSampleTemperature : FB_SampleValue(0, E_OCPP1_ReadingContext.None, E_OCPP1_Measurand.None, E_OCPP1_Phase.None, E_OCPP1_Location.None, E_OCPP1_Unit.None);
	fbSampleVoltageL1 : FB_SampleValue(0, E_OCPP1_ReadingContext.None, E_OCPP1_Measurand.None, E_OCPP1_Phase.None, E_OCPP1_Location.None, E_OCPP1_Unit.None);
	fbSampleVoltageL2 : FB_SampleValue(0, E_OCPP1_ReadingContext.None, E_OCPP1_Measurand.None, E_OCPP1_Phase.None, E_OCPP1_Location.None, E_OCPP1_Unit.None);
	fbSampleVoltageL3 : FB_SampleValue(0, E_OCPP1_ReadingContext.None, E_OCPP1_Measurand.None, E_OCPP1_Phase.None, E_OCPP1_Location.None, E_OCPP1_Unit.None);
	fbSampleFrequency : FB_SampleValue(0, E_OCPP1_ReadingContext.None, E_OCPP1_Measurand.None, E_OCPP1_Phase.None, E_OCPP1_Location.None, E_OCPP1_Unit.None);
END_VAR

METHOD Execute : BOOL
VAR_INPUT
	fbStation : REFERENCE TO FB_Station;
END_VAR
tonSample(
	IN := TRUE,
	PT := VAR_Param.tSampleClock);

fbMeter.Execute();

IF tonSample.Q AND fbStation.Available THEN
	tonSample(IN := FALSE);
	fbSampleTemperature.SetValue(23.4);
	fbSampleVoltageL1.SetValue(230.1);
	fbSampleVoltageL2.SetValue(229.9);
	fbSampleVoltageL3.SetValue(230.0);
	fbSampleFrequency.SetValue(50.012);
	fbMeter.Send();
END_IF
END_METHOD

METHOD FB_Init : BOOL
VAR_INPUT
	bInitRetains : BOOL; // if TRUE, the retain variables are initialized (warm start / cold start)
	bInCopyCode : BOOL;  // if TRUE, the instance afterwards gets moved into the copy code (online change)

	fbStation : REFERENCE TO FB_Station;
END_VAR
IF bInCopyCode THEN RETURN; END_IF

IF NOT __ISVALIDREF(fbStation) THEN RETURN; END_IF

FB_Init := Init(fbStation);
END_METHOD

METHOD Init : BOOL
VAR_IN_OUT CONSTANT
	fbStation : FB_Station;
END_VAR
fbMeter.Init(
	nConnectorId:= 0,
	fbStation:= fbStation);

fbSampleVoltageL1.Init(
	fbMeterValue:= fbMeter,
	eContext:= E_OCPP1_ReadingContext.SampleClock,
	eMeasurand:= E_OCPP1_Measurand.Voltage,
	ePhase:= E_OCPP1_Phase.L1,
	eLocation:= E_OCPP1_Location.None,
	eUnit:= E_OCPP1_Unit.V);

fbSampleVoltageL2.Init(
	fbMeterValue:= fbMeter,
	eContext:= E_OCPP1_ReadingContext.SampleClock,
	eMeasurand:= E_OCPP1_Measurand.Voltage,
	ePhase:= E_OCPP1_Phase.L2,
	eLocation:= E_OCPP1_Location.None,
	eUnit:= E_OCPP1_Unit.V);

fbSampleVoltageL3.Init(
	fbMeterValue:= fbMeter,
	eContext:= E_OCPP1_ReadingContext.SampleClock,
	eMeasurand:= E_OCPP1_Measurand.Voltage,
	ePhase:= E_OCPP1_Phase.L3,
	eLocation:= E_OCPP1_Location.None,
	eUnit:= E_OCPP1_Unit.V);

fbSampleFrequency.Init(
	fbMeterValue:= fbMeter,
	eContext:= E_OCPP1_ReadingContext.SampleClock,
	eMeasurand:= E_OCPP1_Measurand.Frequency,
	ePhase:= E_OCPP1_Phase.None,
	eLocation:= E_OCPP1_Location.None,
	eUnit:= E_OCPP1_Unit.None);
END_METHOD

END_FUNCTION_BLOCK

// ---- POUs/OCPP/FB_MeterValue.TcPOU
FUNCTION_BLOCK FB_MeterValue
VAR
	// id
	_nConnectorId : UDINT;
	// client
	_bSend : BOOL;
	_pClient : POINTER TO FB_OCPP1_Client;
	// sampled values
	_nSampleCnt : UDINT;
	_arrSamples : ARRAY[1..Param_OCPP.nSampledValuesMax] OF POINTER TO FB_SampleValue;
	_arrValues : ARRAY[1..Param_OCPP.nSampledValuesMax] OF ST_OCPP1_SampledValue;
END_VAR

METHOD INTERNAL AddSample : BOOL
VAR_INPUT
	nSampleId : REFERENCE TO UDINT;
	pSample : POINTER TO FB_SampleValue;
END_VAR
IF pSample = 0 THEN
	RETURN; // invalid pointer!
END_IF

IF _nSampleCnt >= Param_OCPP.nSampledValuesMax THEN
	RETURN; // maximum amount of samples!
END_IF

_nSampleCnt := _nSampleCnt + 1;
nSampleId := _nSampleCnt;

_arrSamples[nSampleId] := pSample;

AddSample := TRUE;
END_METHOD

METHOD Execute : BOOL
IF _bSend AND _pClient <> 0 THEN
	IF _pClient^.SendMeterValue(_nConnectorId, _nSampleCnt, _arrValues) THEN
		_bSend := FALSE;
	END_IF
END_IF
END_METHOD

METHOD FB_Init : BOOL
VAR_INPUT
	bInitRetains : BOOL; // if TRUE, the retain variables are initialized (warm start / cold start)
	bInCopyCode : BOOL;  // if TRUE, the instance afterwards gets moved into the copy code (online change)

	nConnectorId : UDINT;
	fbStation : REFERENCE TO FB_Station;
END_VAR
IF bInCopyCode THEN RETURN; END_IF

IF NOT __ISVALIDREF(fbStation) THEN RETURN; END_IF

FB_Init := Init(nConnectorId, fbStation);
END_METHOD

METHOD Init : BOOL
VAR_INPUT
	nConnectorId : UDINT;
END_VAR
VAR_IN_OUT CONSTANT
	fbStation : FB_Station;
END_VAR
_nConnectorId := nConnectorId;

IF __ISVALIDREF(fbStation) THEN
	_pClient := fbStation.Client;
END_IF

Init := (_pClient <> 0);
END_METHOD

METHOD Send : BOOL
VAR
	nIdx : UDINT;
END_VAR
IF _pClient = 0 THEN
	RETURN; // invalid pointer to client!
END_IF

IF NOT _bSend THEN
	FOR nIdx := 1 TO _nSampleCnt DO
		IF _arrSamples[nIdx] <> 0 THEN
			_arrSamples[nIdx]^.GetSampled(_arrValues[nIdx]);
		END_IF
	END_FOR
	_bSend := TRUE;
END_IF

IF _pClient <> 0 THEN
	Send := _pClient^.SendMeterValue(_nConnectorId, _nSampleCnt, _arrValues);
	IF Send THEN _bSend := FALSE; END_IF
END_IF
END_METHOD

END_FUNCTION_BLOCK

// ---- POUs/OCPP/FB_SampleValue.TcPOU
FUNCTION_BLOCK FB_SampleValue
VAR
	_nSampleId : UDINT;
	_mValue : ST_OCPP1_SampledValue;
END_VAR

METHOD FB_Init : BOOL
VAR_INPUT
	bInitRetains : BOOL; // if TRUE, the retain variables are initialized (warm start / cold start)
	bInCopyCode : BOOL;  // if TRUE, the instance afterwards gets moved into the copy code (online change)

	fbMeterValue : REFERENCE TO FB_MeterValue;
	eContext : E_OCPP1_ReadingContext := E_OCPP1_ReadingContext.SamplePeriodic; // Optional. Type of detail value: start, end or sample.
	eMeasurand : E_OCPP1_Measurand := E_OCPP1_Measurand.None; // Optional. Type of measurement.
	ePhase : E_OCPP1_Phase := E_OCPP1_Phase.None; // Optional. indicates how the measured value is to be interpreted.
	eLocation : E_OCPP1_Location := E_OCPP1_Location.None; // Optional. Location of measurement.
	eUnit : E_OCPP1_Unit := E_OCPP1_Unit.None; // Optional. Unit of the value.
END_VAR
IF bInCopyCode THEN RETURN; END_IF

IF NOT __ISVALIDREF(fbMeterValue) THEN RETURN; END_IF

FB_Init := Init(fbMeterValue, eContext, eMeasurand, ePhase, eLocation, eUnit);
END_METHOD

METHOD INTERNAL GetSampled : BOOL
VAR_IN_OUT
	mSampledValue : ST_OCPP1_SampledValue;
END_VAR
mSampledValue := _mValue;
END_METHOD

METHOD Init : BOOL
VAR_INPUT
	fbMeterValue : REFERENCE TO FB_MeterValue;
	eContext : E_OCPP1_ReadingContext := E_OCPP1_ReadingContext.SamplePeriodic; // Optional. Type of detail value: start, end or sample.
	eMeasurand : E_OCPP1_Measurand := E_OCPP1_Measurand.None; // Optional. Type of measurement.
	ePhase : E_OCPP1_Phase := E_OCPP1_Phase.None; // Optional. indicates how the measured value is to be interpreted.
	eLocation : E_OCPP1_Location := E_OCPP1_Location.None; // Optional. Location of measurement.
	eUnit : E_OCPP1_Unit := E_OCPP1_Unit.None; // Optional. Unit of the value.
END_VAR
_mValue.fValue := 0.0;
_mValue.eContext := eContext;
_mValue.eMeasurand := eMeasurand;
_mValue.ePhase := ePhase;
_mValue.eLocation := eLocation;
_mValue.eUnit := eUnit;

Init := fbMeterValue.AddSample(_nSampleId, THIS);
END_METHOD

METHOD SetValue : BOOL
VAR_INPUT
	fValue : LREAL;
END_VAR
_mValue.fValue := fValue;
END_METHOD

PROPERTY Value : LREAL
GET
Value := _mValue.fValue;
END_GET
SET
_mValue.fValue := Value;
END_SET
END_PROPERTY

END_FUNCTION_BLOCK

// ---- POUs/OCPP/FB_ConnectorMeter.TcPOU
FUNCTION_BLOCK FB_ConnectorMeter
VAR
	tonSample : TON;
	fbMeter : FB_MeterValue(0, 0);
	fbSampleEnergy : FB_SampleValue(0, E_OCPP1_ReadingContext.None, E_OCPP1_Measurand.None, E_OCPP1_Phase.None, E_OCPP1_Location.None, E_OCPP1_Unit.None);
	fbSampleCurrentL1 : FB_SampleValue(0, E_OCPP1_ReadingContext.None, E_OCPP1_Measurand.None, E_OCPP1_Phase.None, E_OCPP1_Location.None, E_OCPP1_Unit.None);
	fbSampleCurrentL2 : FB_SampleValue(0, E_OCPP1_ReadingContext.None, E_OCPP1_Measurand.None, E_OCPP1_Phase.None, E_OCPP1_Location.None, E_OCPP1_Unit.None);
	fbSampleCurrentL3 : FB_SampleValue(0, E_OCPP1_ReadingContext.None, E_OCPP1_Measurand.None, E_OCPP1_Phase.None, E_OCPP1_Location.None, E_OCPP1_Unit.None);
	fbSamplePower : FB_SampleValue(0, E_OCPP1_ReadingContext.None, E_OCPP1_Measurand.None, E_OCPP1_Phase.None, E_OCPP1_Location.None, E_OCPP1_Unit.None);
END_VAR

METHOD Execute : BOOL
VAR_INPUT
	fbConnector : REFERENCE TO FB_Connector;
	fCurrentOffered : REAL; // [A]
END_VAR
tonSample(
	IN := fbConnector.bCharging,
	PT := VAR_Param.tSamplePeriodic);

fbMeter.Execute();

IF tonSample.Q AND fbConnector.Available THEN
	tonSample(IN := FALSE);
	fbSampleEnergy.SetValue(fbConnector.nEnergyMeter);
	fbSampleCurrentL1.SetValue(fCurrentOffered);
	fbSampleCurrentL2.SetValue(fCurrentOffered);
	fbSampleCurrentL3.SetValue(fCurrentOffered);
	fbSamplePower.SetValue(fCurrentOffered * 3.0 * 230.0 * 0.001);
	fbMeter.Send();
END_IF
END_METHOD

METHOD FB_Init : BOOL
VAR_INPUT
	bInitRetains : BOOL; // if TRUE, the retain variables are initialized (warm start / cold start)
	bInCopyCode : BOOL;  // if TRUE, the instance afterwards gets moved into the copy code (online change)

	nConnectorId : UDINT;
	fbStation : REFERENCE TO FB_Station;
END_VAR
IF bInCopyCode THEN RETURN; END_IF

IF NOT __ISVALIDREF(fbStation) THEN RETURN; END_IF

FB_Init := Init(nConnectorId, fbStation);
END_METHOD

METHOD Init : BOOL
VAR_INPUT
	nConnectorId : UDINT;
	fbStation : REFERENCE TO FB_Station;
END_VAR
fbMeter.Init(
	nConnectorId:= nConnectorId,
	fbStation:= fbStation);

fbSampleEnergy.Init(
	fbMeterValue:= fbMeter,
	eContext:= E_OCPP1_ReadingContext.SamplePeriodic,
	eMeasurand:= E_OCPP1_Measurand.EnergyActiveImportRegister,
	ePhase:= E_OCPP1_Phase.None,
	eLocation:= E_OCPP1_Location.None,
	eUnit:= E_OCPP1_Unit.Wh);

fbSampleCurrentL1.Init(
	fbMeterValue:= fbMeter,
	eContext:= E_OCPP1_ReadingContext.SamplePeriodic,
	eMeasurand:= E_OCPP1_Measurand.CurrentImport,
	ePhase:= E_OCPP1_Phase.L1,
	eLocation:= E_OCPP1_Location.None,
	eUnit:= E_OCPP1_Unit.A);

fbSampleCurrentL2.Init(
	fbMeterValue:= fbMeter,
	eContext:= E_OCPP1_ReadingContext.SamplePeriodic,
	eMeasurand:= E_OCPP1_Measurand.CurrentImport,
	ePhase:= E_OCPP1_Phase.L2,
	eLocation:= E_OCPP1_Location.None,
	eUnit:= E_OCPP1_Unit.A);

fbSampleCurrentL3.Init(
	fbMeterValue:= fbMeter,
	eContext:= E_OCPP1_ReadingContext.SamplePeriodic,
	eMeasurand:= E_OCPP1_Measurand.CurrentImport,
	ePhase:= E_OCPP1_Phase.L3,
	eLocation:= E_OCPP1_Location.None,
	eUnit:= E_OCPP1_Unit.A);

fbSamplePower.Init(
	fbMeterValue:= fbMeter,
	eContext:= E_OCPP1_ReadingContext.SamplePeriodic,
	eMeasurand:= E_OCPP1_Measurand.PowerActiveImport,
	ePhase:= E_OCPP1_Phase.None,
	eLocation:= E_OCPP1_Location.None,
	eUnit:= E_OCPP1_Unit.kW);
END_METHOD

END_FUNCTION_BLOCK

// ---- POUs/FB_ConnectorSim.TcPOU
FUNCTION_BLOCK FB_ConnectorSim
VAR_INPUT
	sIdTag : T_OCPP1_IdToken := '1234abcd';
	bAuto : BOOL; // automatic start/stop of charging
	bAuth : BOOL; // authorize token (e.g. from RFID)
	bPlug : BOOL; // cable from EV connected to EVSE
	bStart : BOOL; // start transaction for charging
	bStop : BOOL; // stop transaction of charging
	fCurrentOffered : REAL; // [A] limitation of offered current
	tWaitStart : TIME := T#1M10S; // wait time to start transaction in auto mode
	tWaitCharge : TIME := T#3M45S; // wait time to charge and stop transaction in auto mode
END_VAR
VAR_IN_OUT
	fbConnector : FB_Connector;
END_VAR
VAR
	nState : BYTE;
	tonDelay : TON;
	tonLocked : TON;
	tonOffering : TON;
	tonCharging : TON;
	trigDisconnect : F_TRIG;
	fPowerOffered : REAL; // [W]
END_VAR
VAR PERSISTENT
	fEnergyMeterIntegrator : REAL; // [Wh] meter value of charged energy
END_VAR

CASE nState OF
	0: // init => wait
		IF bAuto THEN
			tonDelay(IN := FALSE);
			nState := 1;
		END_IF
	1: // wait => start
		tonDelay(IN := TRUE, PT := tWaitStart);
		IF tonDelay.Q THEN
			bPlug := TRUE;
			bStart := TRUE;
			tonDelay(IN := FALSE);
			nState := 2;
		END_IF
	2: // charge => stop
		tonDelay(IN := TRUE, PT := tWaitCharge);
		IF tonDelay.Q THEN
			bPlug := FALSE;
			bStop := TRUE;
			tonDelay(IN := FALSE);
			nState := 1;
		END_IF
ELSE
	nState := 0;
END_CASE

fbConnector.bOperative := TRUE;
fbConnector.sIdTag := sIdTag;

fbConnector.bAuth := bAuth;
fbConnector.bConnected := bPlug;
fbConnector.bStart := bStart;
fbConnector.bStop := bStop;

tonLocked(IN := fbConnector.bLock, PT := T#500MS, Q => fbConnector.bLocked);
tonOffering(IN := fbConnector.bSupply, PT := T#500MS, Q => fbConnector.bOffering);
tonCharging(IN := fbConnector.bSupply, PT := T#2S, Q => fbConnector.bCharging);

IF fCurrentOffered > fbConnector.fChargeLimit THEN
	fCurrentOffered := fbConnector.fChargeLimit; // [A] limited by charging profile
END_IF

IF tonCharging.Q THEN
	fPowerOffered := fCurrentOffered * 3.0 * 230.0 / 3600.0; // [W/s] charging power at three phases with 230V
	fEnergyMeterIntegrator := fEnergyMeterIntegrator + fPowerOffered * 0.01; // [Wh] charging energy meter at 10ms cycle time
	fbConnector.nEnergyMeter := LREAL_TO_UDINT(fEnergyMeterIntegrator);
END_IF

trigDisconnect(CLK := fbConnector.bLock);
IF trigDisconnect.Q THEN
	fbConnector.bConnected := FALSE;
END_IF

bAuth := FALSE;
IF bStart AND fbConnector.bCharging THEN
	bStart := FALSE;
END_IF
IF bStop AND NOT fbConnector.bCharging THEN
	bStop := FALSE;
END_IF

END_FUNCTION_BLOCK
